// TIA Portal V19 export
TYPE "Prg_GetITF"
// stored: Access Published
   STRUCT
      PrgNo : DInt;
      Execute : Bool;
      InProgress : Bool;
      Done : Bool;
      Error : Bool;
   END_STRUCT;
END_TYPE
